// TIA Portal V19 export
FUNCTION "AddTwo" : Void   // FC0, SCL
BEGIN
   #AddTwo := #a + #b;
END_FUNCTION
